// TIA Portal project "final code of X Y  plotter 31may2023" (V17)

(* hardware
DEVICE "S7-1200 station_1"  S7-1200 Station
   slot 0: "Rack_0"  S7-1200 Rack  Rack  V1.0
   slot 1: "PLC_1"  CPU 1214C DC/DC/DC  6ES7 214-1AG40-0XB0  V4.5
*)

// ===== PLC "PLC_1"  CPU 1214C DC/DC/DC =====

VAR_GLOBAL   // PLC tag table "Default tag table"
   "Axis_1_LowHwLimitSwitch" AT %I0.3 : Bool;
   "Axis_1_HighHwLimitSwitch" AT %I0.4 : Bool;
   "Axis_1_Homing switch" AT %I1.3 : Bool;
   "Axis_2_LowHwLimitSwitch" AT %I1.0 : Bool;
   "Axis_2_HighHwLimitSwitch" AT %I1.1 : Bool;
   "Axis_2_Homing switch" AT %I1.2 : Bool;
   "Homing" AT %I0.5 : Bool;
   "push button 3" AT %I0.0 : Bool;
   "Not in use" AT %I0.1 : Bool;
   "push button 2" AT %I0.2 : Bool;
   "Switch" AT %I0.7 : Bool;
   "Selector_SW_1" AT %I8.1 : Bool;
   "Selector_SW_2" AT %I8.2 : Bool;
   "Selector_SW_3" AT %I8.3 : Bool;
   "Selector_SW_4" AT %I8.4 : Bool;
   "ABS SWITCH Continue" AT %I1.5 : Bool;
   "reset_switch" AT %I0.6 : Bool;
   "X axis Encoder Readings" AT %ID1000 : Real;
   "Y axis Encoder Readings" AT %ID1004 : Real;
   "Axis_1_Pulse" AT %Q0.0 : Bool;
   "Axis_1_Direction" AT %Q0.5 : Bool;
   "Axis_2_Direction" AT %Q0.7 : Bool;
   "Solnoid" AT %Q1.1 : Bool;
   "Axis_2_Pulse" AT %Q0.2 : Bool;
   "X_axis_pw_error" AT %M100.0 : Bool;
   "X_axis_pw_error_1" AT %M100.1 : Bool;
   "X_axis_pw_delay" AT %M100.2 : Bool;
   "Y_axis_pw_error" AT %M100.3 : Bool;
   "Y_axis_pw_error_1" AT %M100.4 : Bool;
   "Y_axis_pw_delay" AT %M100.5 : Bool;
   "X_AXIS_HOME_DONE" AT %M0.1 : Bool;
   "Y_AXIS_HOME_DONE" AT %M0.2 : Bool;
   "Y_Position" AT %MD104 : Real;
   "X_Velosity" AT %MD112 : Real;
   "Y_Velosity" AT %MD116 : Real;
   "X_Position" AT %MD120 : Real;
   "Y_Abs_DONE" AT %M101.4 : Bool;
   "X_Abs_DONE" AT %M101.3 : Bool;
   "X_done" AT %MD124 : Real;
   "Y_done" AT %MD128 : Real;
   "X_AXIS_HOME_DONE_latch" AT %M0.3 : Bool;
   "Y_AXIS_HOME_DONE_latch" AT %M0.4 : Bool;
   "Homing_TON_IN" AT %M0.5 : Bool;
   "X_AXIS_ABS_BUSY" AT %M0.6 : Bool;
   "Y_AXIS_ABS_BUSY" AT %M0.7 : Bool;
   "Homing_TON_OUT" AT %M6.0 : Bool;
   "X_AXIS_HOME_DN_LATCH" AT %M10.0 : Bool;
   "Y_AXIS_HOME_DN_LATCH" AT %M10.1 : Bool;
   "MC_HOME_DN" AT %M10.2 : Bool;
   "h_done" AT %MD140 : Real;
   "X_AXIS_ABS_DN" AT %M11.1 : Bool;
   "Y_AXIS_ABS_DN" AT %M11.2 : Bool;
   "MC_ABS_DN" AT %M11.3 : Bool;
   "NEXT_ABS_EXE" AT %MD144 : Real;
   "Prev_X_VAL" AT %MD156 : Real;
   "Prev_X_To_Program" AT %MD148 : Real;
   "Prev_Y_VAL" AT %MD160 : Real;
   "Prev_Y_To_Program" AT %MD152 : Real;
   "Sol_Cmd_from python" AT %MD164 : Real;
   "GG_BIT from python code" AT %MD200 : Real;
   "To_g_stat" AT %M7.6 : Bool;
   "g_stat" AT %MD212 : Real;
   "g_stat_plc" AT %MD216 : Real;
   "g_stat_1" AT %M8.1 : Bool;
   "g_stat_latch" AT %M8.2 : Bool;
   "Abs_dn_latch" AT %M8.4 : Bool;
   "X1_done" AT %MD220 : Real;
   "Y1_done" AT %MD224 : Real;
   "ABS_BUTTON" AT %MD108 : Real;
   "X Encoder" AT %MD228 : Real;
   "Y Encoder" AT %MD232 : Real;
   "X Encoder ABS" AT %MD236 : Real;
   "X Encoder Multiplier" AT %MD240 : Real;
   "X AxisActual pos" AT %MD244 : Real;
   "Y AxisActual pos" AT %MD248 : Real;
   "Homing Function from front end" AT %MD252 : Real;
   "Softbit_homing" AT %M12.0 : Bool;
END_VAR

TYPE "User_data_type_1"
VERSION : 0.1
   STRUCT
      "HR location" : Int;
   END_STRUCT;
END_TYPE

// folder: System blocks/Program resources

DATA_BLOCK "IEC_Timer_0_DB"   // DB6
{ S7_Optimized_Access := 'TRUE' }
AUTHOR : Simatic
FAMILY : IEC
NAME : IEC_TMR
VERSION : 1.0
// stored: InstanceOfName IEC_TIMER
"IEC_TIMER"
BEGIN
END_DATA_BLOCK

DATA_BLOCK "IEC_Timer_0_DB_2"   // DB11
{ S7_Optimized_Access := 'TRUE' }
AUTHOR : Simatic
FAMILY : IEC
NAME : IEC_TMR
VERSION : 1.0
// stored: InstanceOfName IEC_TIMER
"IEC_TIMER"
BEGIN
END_DATA_BLOCK

DATA_BLOCK "IEC_Timer_0_DB_1"   // DB13
{ S7_Optimized_Access := 'TRUE' }
AUTHOR : Simatic
FAMILY : IEC
NAME : IEC_TMR
VERSION : 1.0
// stored: InstanceOfName IEC_TIMER
"IEC_TIMER"
BEGIN
END_DATA_BLOCK

// folder: (top level)

DATA_BLOCK "Axis_1"   // DB1, Motion_DB
{ S7_Optimized_Access := 'TRUE' }
AUTHOR : SIMATIC
FAMILY : BasicMC
NAME : TO_PosAx
VERSION : 8.0
// stored: InstanceOfName TO_PositioningAxis
"TO_PositioningAxis"
BEGIN
   // Axis.LengthUnitNormalized.Distance = 1013
   // Axis.HomingReferencePointSwitch_AddressCU = %I1.3
   // Axis.PositionLimitsMax_AddressCU = %I0.4
   // Axis.PositionLimitsMin_AddressCU = %I0.3
   // Axis.OnlinePtoModeCU = 16#0000_0002
   // Axis.DirectionOutputEnabledCU = TRUE
   // Axis.SelectedChannel2EnumCU = %Q0.5
   // Axis.SelectedChannel1EnumCU = %Q0.0
   // Pulse.MinDeltaDeltaFrequencyCU = 0.004
   // Pulse.MaxDeltaDeltaFrequencyCU = 1.0E+10
   // Pulse.MinDeltaFrequencyCU = 0.005
   // Pulse.MaxDeltaFrequencyCU = 9.5E+9
   // Pulse.MinFrequencyCU = 1.0
   // Pulse.MaxFrequencyCU = 100000.0
   // Pulse.OutputSourceCU = 16#0000_0000
   // Axis.SelectPTO = 0
END_DATA_BLOCK

DATA_BLOCK "Axis_2"   // DB2, Motion_DB
{ S7_Optimized_Access := 'TRUE' }
AUTHOR : SIMATIC
FAMILY : BasicMC
NAME : TO_PosAx
VERSION : 8.0
// stored: InstanceOfName TO_PositioningAxis
"TO_PositioningAxis"
BEGIN
   // Axis.HomingReferencePointSwitch_AddressCU = %I1.2
   // Axis.PositionLimitsMax_AddressCU = %I1.1
   // Axis.PositionLimitsMin_AddressCU = %I1.0
   // Axis.LengthUnitNormalized.Distance = 1013
   // Axis.DirectionOutputEnabledCU = TRUE
   // Axis.OnlinePtoModeCU = 16#0000_0002
   // Axis.SelectedChannel2EnumCU = %Q0.7
   // Axis.SelectedChannel1EnumCU = %Q0.2
   // Pulse.MinDeltaDeltaFrequencyCU = 0.004
   // Pulse.MaxDeltaDeltaFrequencyCU = 1.0E+10
   // Pulse.MinDeltaFrequencyCU = 0.005
   // Pulse.MaxDeltaFrequencyCU = 9.5E+9
   // Pulse.MinFrequencyCU = 1.0
   // Pulse.MaxFrequencyCU = 100000.0
   // Pulse.OutputSourceCU = 16#0000_0000
   // Axis.SelectPTO = 1
   // Axis.OnlinePtoIndexCU = 1
END_DATA_BLOCK

DATA_BLOCK "Command table_X"   // DB28, BMC_202
{ S7_Optimized_Access := 'TRUE' }
AUTHOR : SIMATIC
FAMILY : BasicMC
NAME : CmdTab
VERSION : 8.0
// stored: InstanceOfName TO_CommandTable
"TO_CommandTable"
BEGIN
   // BasicMotionControl.CompileUnit.ExtendedGeneral.ConnectedAxisDBName = Axis_1
   // BasicMotionControl.CompileUnit.ExtendedGeneral.UsedParameters = 1
   // BasicMotionControl.CompileUnit.ExtendedGeneral.AxisID = {2232340-7248}
END_DATA_BLOCK

DATA_BLOCK "Command table_Y"   // DB29, BMC_202
{ S7_Optimized_Access := 'TRUE' }
AUTHOR : SIMATIC
FAMILY : BasicMC
NAME : CmdTab
VERSION : 8.0
// stored: InstanceOfName TO_CommandTable
"TO_CommandTable"
BEGIN
   // BasicMotionControl.CompileUnit.ExtendedGeneral.ConnectedAxisDBName = Axis_2
   // BasicMotionControl.CompileUnit.ExtendedGeneral.UsedParameters = 2
   // BasicMotionControl.CompileUnit.ExtendedGeneral.AxisID = {2232340-2021}
END_DATA_BLOCK

ORGANIZATION_BLOCK "Main"   // OB1, LAD, ProgramCycle
TITLE = "Main Program Sweep (Cycle)"
{ S7_Optimized_Access := 'TRUE' }
VERSION : 0.1
   VAR_INPUT
      Initial_Call : Bool;   // Initial call of this OB
      Remanence : Bool;   // =True, if remanent data are available
   END_VAR
BEGIN

REGION Network 1: POWER
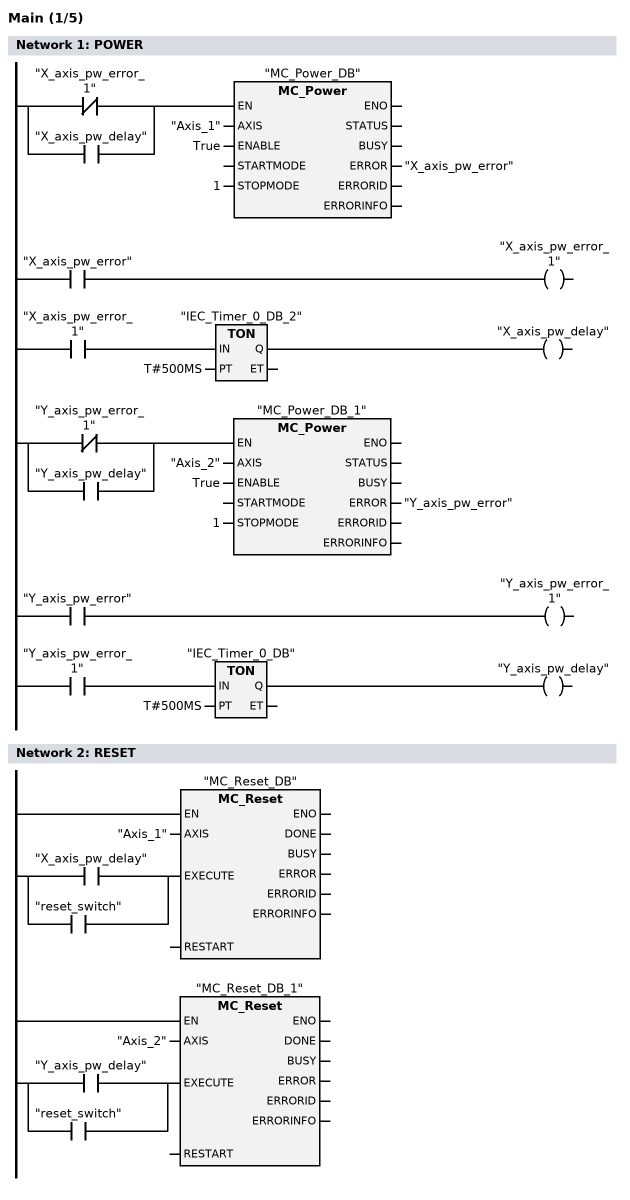
   IF NOT "X_axis_pw_error_1" OR "X_axis_pw_delay" THEN
       "MC_Power_DB"(Axis := "Axis_1", Enable := True, StopMode := 1, Error => "X_axis_pw_error");   // MC_Power
   END_IF;
   "X_axis_pw_error_1" := "X_axis_pw_error";
   "IEC_Timer_0_DB_2".TON(IN := "X_axis_pw_error_1", PT := T#500MS);
   "X_axis_pw_delay" := "IEC_Timer_0_DB_2".Q;
   IF NOT "Y_axis_pw_error_1" OR "Y_axis_pw_delay" THEN
       "MC_Power_DB_1"(Axis := "Axis_2", Enable := True, StopMode := 1, Error => "Y_axis_pw_error");   // MC_Power
   END_IF;
   "Y_axis_pw_error_1" := "Y_axis_pw_error";
   "IEC_Timer_0_DB".TON(IN := "Y_axis_pw_error_1", PT := T#500MS);
   "Y_axis_pw_delay" := "IEC_Timer_0_DB".Q;
END_REGION

REGION Network 2: RESET
   "MC_Reset_DB"(Axis := "Axis_1", Execute := "X_axis_pw_delay" OR "reset_switch");   // MC_Reset
   "MC_Reset_DB_1"(Axis := "Axis_2", Execute := "Y_axis_pw_delay" OR "reset_switch");   // MC_Reset
END_REGION

REGION Network 3: HOME
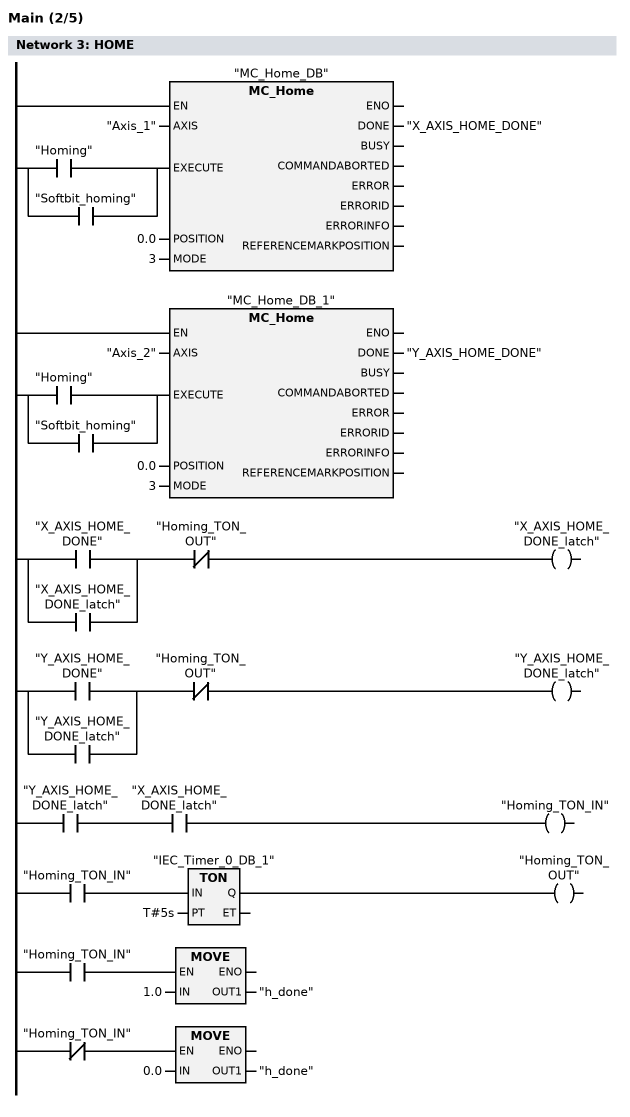
   "MC_Home_DB"(Axis := "Axis_1",   // MC_Home
                Execute := "Homing" OR "Softbit_homing",
                Position := 0.0,
                Mode := 3,
                Done => "X_AXIS_HOME_DONE");
   "MC_Home_DB_1"(Axis := "Axis_2",   // MC_Home
                  Execute := "Homing" OR "Softbit_homing",
                  Position := 0.0,
                  Mode := 3,
                  Done => "Y_AXIS_HOME_DONE");
   "X_AXIS_HOME_DONE_latch" := ("X_AXIS_HOME_DONE" OR "X_AXIS_HOME_DONE_latch") AND NOT "Homing_TON_OUT";
   "Y_AXIS_HOME_DONE_latch" := ("Y_AXIS_HOME_DONE" OR "Y_AXIS_HOME_DONE_latch") AND NOT "Homing_TON_OUT";
   "Homing_TON_IN" := "Y_AXIS_HOME_DONE_latch" AND "X_AXIS_HOME_DONE_latch";
   "IEC_Timer_0_DB_1".TON(IN := "Homing_TON_IN", PT := T#5s);
   "Homing_TON_OUT" := "IEC_Timer_0_DB_1".Q;
   IF "Homing_TON_IN" THEN "h_done" := 1.0; END_IF;
   IF NOT "Homing_TON_IN" THEN "h_done" := 0.0; END_IF;
END_REGION

REGION Network 4: Absolute
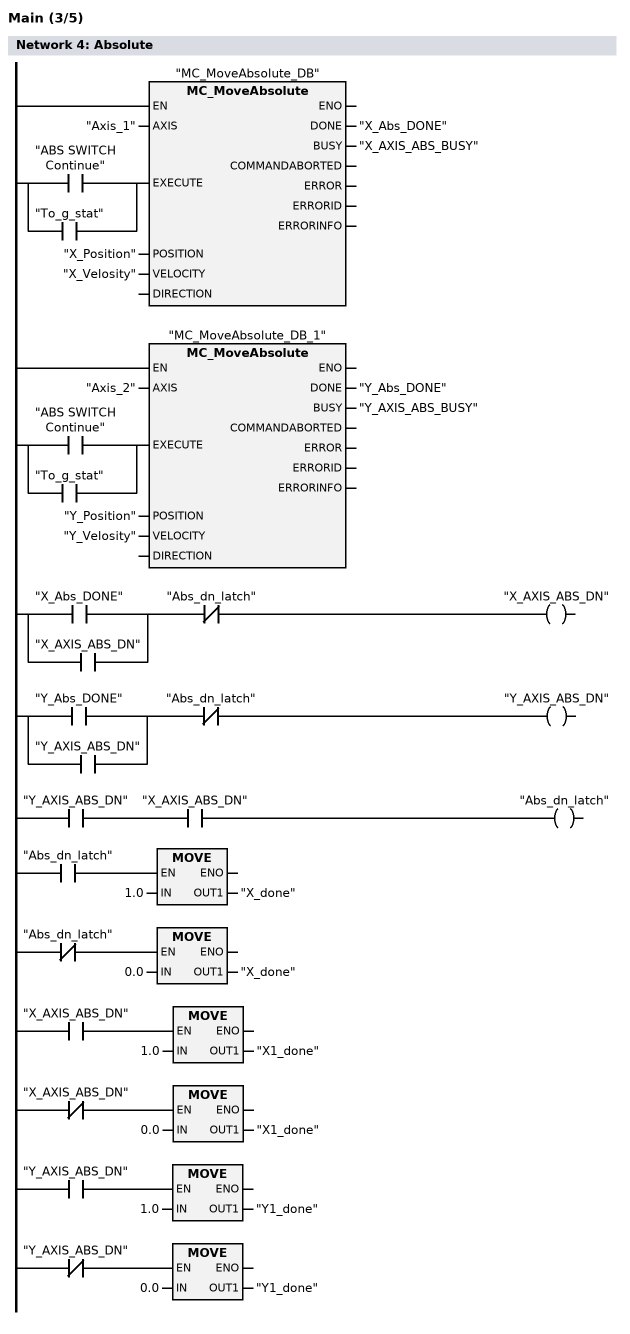
   "MC_MoveAbsolute_DB"(Axis := "Axis_1",   // MC_MoveAbsolute
                        Execute := "ABS SWITCH Continue" OR "To_g_stat",
                        Position := "X_Position",
                        Velocity := "X_Velosity",
                        Done => "X_Abs_DONE",
                        Busy => "X_AXIS_ABS_BUSY");
   "MC_MoveAbsolute_DB_1"(Axis := "Axis_2",   // MC_MoveAbsolute
                          Execute := "ABS SWITCH Continue" OR "To_g_stat",
                          Position := "Y_Position",
                          Velocity := "Y_Velosity",
                          Done => "Y_Abs_DONE",
                          Busy => "Y_AXIS_ABS_BUSY");
   "X_AXIS_ABS_DN" := ("X_Abs_DONE" OR "X_AXIS_ABS_DN") AND NOT "Abs_dn_latch";
   "Y_AXIS_ABS_DN" := ("Y_Abs_DONE" OR "Y_AXIS_ABS_DN") AND NOT "Abs_dn_latch";
   "Abs_dn_latch" := "Y_AXIS_ABS_DN" AND "X_AXIS_ABS_DN";
   IF "Abs_dn_latch" THEN "X_done" := 1.0; END_IF;
   IF NOT "Abs_dn_latch" THEN "X_done" := 0.0; END_IF;
   IF "X_AXIS_ABS_DN" THEN "X1_done" := 1.0; END_IF;
   IF NOT "X_AXIS_ABS_DN" THEN "X1_done" := 0.0; END_IF;
   IF "Y_AXIS_ABS_DN" THEN "Y1_done" := 1.0; END_IF;
   IF NOT "Y_AXIS_ABS_DN" THEN "Y1_done" := 0.0; END_IF;
END_REGION

REGION Network 5
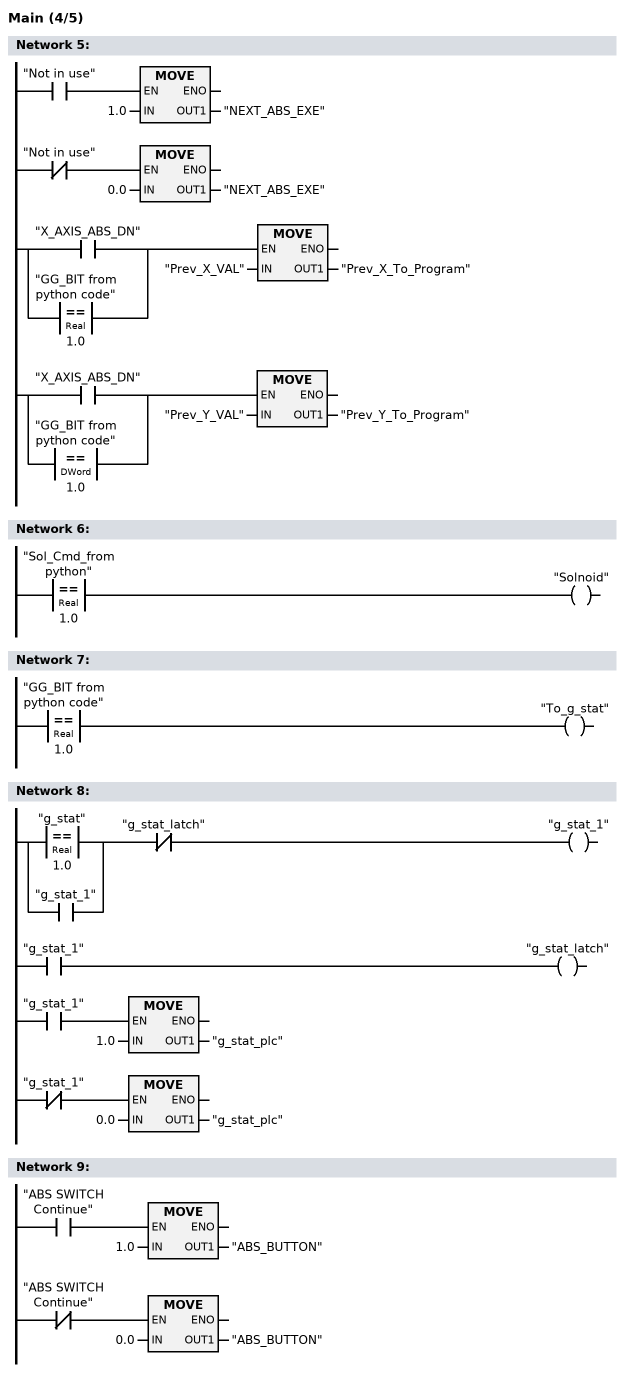
   RUNG wire#powerrail
      Contact( "Not in use" )
      Move(in := 1.0, out1 => "NEXT_ABS_EXE")
   END_RUNG
   RUNG wire#powerrail
      I_Contact( "Not in use" )
      Move(in := 0.0, out1 => "NEXT_ABS_EXE")
   END_RUNG
   RUNG wire#powerrail
      Contact( "X_AXIS_ABS_DN" )
      wire#w1
      Move(in := "Prev_X_VAL", out1 => "Prev_X_To_Program")
   END_RUNG
   RUNG wire#powerrail
      { S7_Templates := "SrcType := Real" } EQ_Contact(in1 := "GG_BIT from python code", in2 := 1.0)
   END_RUNG wire#w1
   RUNG wire#powerrail
      Contact( "X_AXIS_ABS_DN" )
      wire#w2
      Move(in := "Prev_Y_VAL", out1 => "Prev_Y_To_Program")
   END_RUNG
   RUNG wire#powerrail
      { S7_Templates := "SrcType := DWord" } EQ_Contact(in1 := "GG_BIT from python code", in2 := 1.0)
   END_RUNG wire#w2
   // the same network as SCL:
   IF "Not in use" THEN "NEXT_ABS_EXE" := 1.0; END_IF;
   IF NOT "Not in use" THEN "NEXT_ABS_EXE" := 0.0; END_IF;
   IF "X_AXIS_ABS_DN" OR ("GG_BIT from python code" = 1.0) THEN
       "Prev_X_To_Program" := "Prev_X_VAL";
       "Prev_Y_To_Program" := "Prev_Y_VAL";
   END_IF;
END_REGION

REGION Network 6
   RUNG wire#powerrail
      { S7_Templates := "SrcType := Real" } EQ_Contact(in1 := "Sol_Cmd_from python", in2 := 1.0)
      Coil( "Solnoid" )
   END_RUNG
   // the same network as SCL:
   "Solnoid" := "Sol_Cmd_from python" = 1.0;
END_REGION

REGION Network 7
   RUNG wire#powerrail
      { S7_Templates := "SrcType := Real" } EQ_Contact(in1 := "GG_BIT from python code", in2 := 1.0)
      Coil( "To_g_stat" )
   END_RUNG
   // the same network as SCL:
   "To_g_stat" := "GG_BIT from python code" = 1.0;
END_REGION

REGION Network 8
   RUNG wire#powerrail
      { S7_Templates := "SrcType := Real" } EQ_Contact(in1 := "g_stat", in2 := 1.0)
      wire#w1
      I_Contact( "g_stat_latch" )
      Coil( "g_stat_1" )
   END_RUNG
   RUNG wire#powerrail
      Contact( "g_stat_1" )
   END_RUNG wire#w1
   RUNG wire#powerrail
      Contact( "g_stat_1" )
      Coil( "g_stat_latch" )
   END_RUNG
   RUNG wire#powerrail
      Contact( "g_stat_1" )
      Move(in := 1.0, out1 => "g_stat_plc")
   END_RUNG
   RUNG wire#powerrail
      I_Contact( "g_stat_1" )
      Move(in := 0.0, out1 => "g_stat_plc")
   END_RUNG
   // the same network as SCL:
   "g_stat_1" := (("g_stat" = 1.0) OR "g_stat_1") AND NOT "g_stat_latch";
   "g_stat_latch" := "g_stat_1";
   IF "g_stat_1" THEN "g_stat_plc" := 1.0; END_IF;
   IF NOT "g_stat_1" THEN "g_stat_plc" := 0.0; END_IF;
END_REGION

REGION Network 9
   RUNG wire#powerrail
      Contact( "ABS SWITCH Continue" )
      Move(in := 1.0, out1 => "ABS_BUTTON")
   END_RUNG
   RUNG wire#powerrail
      I_Contact( "ABS SWITCH Continue" )
      Move(in := 0.0, out1 => "ABS_BUTTON")
   END_RUNG
   // the same network as SCL:
   IF "ABS SWITCH Continue" THEN "ABS_BUTTON" := 1.0; END_IF;
   IF NOT "ABS SWITCH Continue" THEN "ABS_BUTTON" := 0.0; END_IF;
END_REGION

REGION Network 10: Encoder
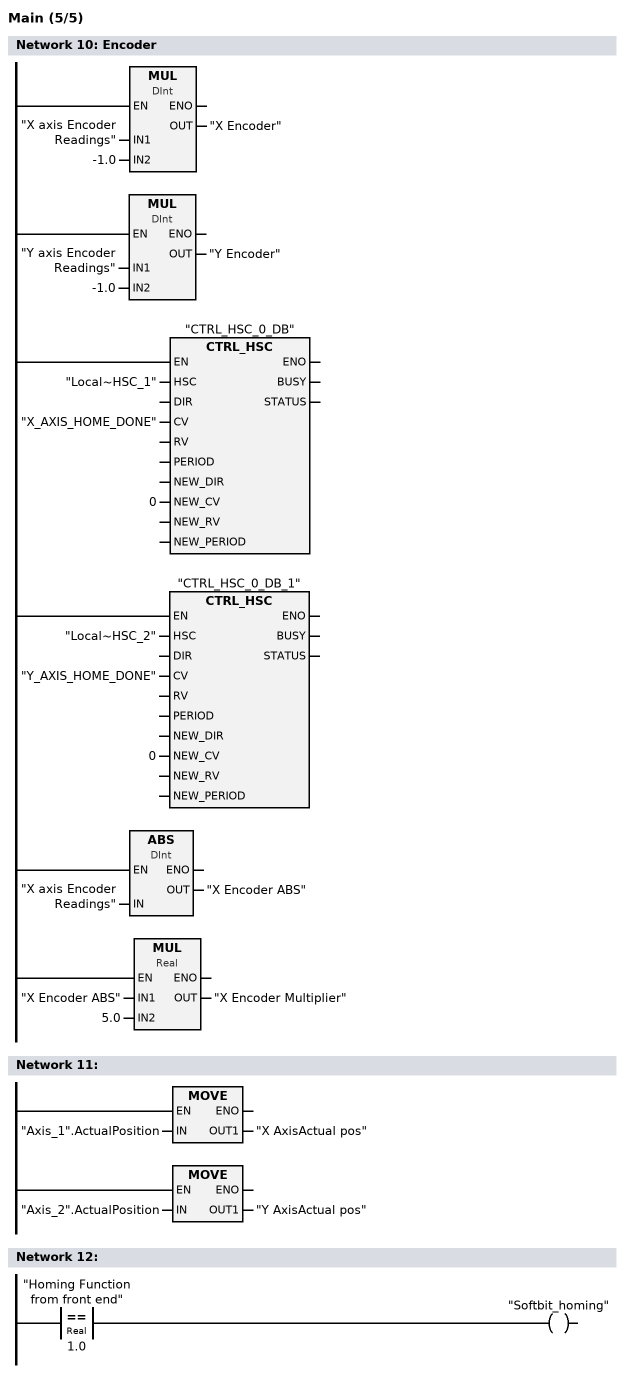
   "X Encoder" := "X axis Encoder Readings" * (-1.0);
   "Y Encoder" := "Y axis Encoder Readings" * (-1.0);
   "CTRL_HSC_0_DB"(HSC := "Local~HSC_1", CV := "X_AXIS_HOME_DONE", NEW_CV := 0);   // CTRL_HSC
   "CTRL_HSC_0_DB_1"(HSC := "Local~HSC_2", CV := "Y_AXIS_HOME_DONE", NEW_CV := 0);   // CTRL_HSC
   "X Encoder ABS" := ABS("X axis Encoder Readings");
   "X Encoder Multiplier" := "X Encoder ABS" * 5.0;
END_REGION

REGION Network 11
   RUNG wire#powerrail
      Move(in := "Axis_1".ActualPosition, out1 => "X AxisActual pos")
   END_RUNG
   RUNG wire#powerrail
      Move(in := "Axis_2".ActualPosition, out1 => "Y AxisActual pos")
   END_RUNG
   // the same network as SCL:
   "X AxisActual pos" := "Axis_1".ActualPosition;
   "Y AxisActual pos" := "Axis_2".ActualPosition;
END_REGION

REGION Network 12
   RUNG wire#powerrail
      { S7_Templates := "SrcType := Real" } EQ_Contact(in1 := "Homing Function from front end", in2 := 1.0)
      Coil( "Softbit_homing" )
   END_RUNG
   // the same network as SCL:
   "Softbit_homing" := "Homing Function from front end" = 1.0;
END_REGION
END_ORGANIZATION_BLOCK